Staubli VAL3: ToolItem.pjx

--- ToolItem.pjx ---
Parameters version=s7.2.1 stackSize=5000 millimeterUnit=true
Data file=toolItem.dtx
Type name=InstrItem path=Disk://kernel/template/InstrItem/InstrItem.pjx

--- ToolItem.dtx ---
public InstrItem iActionOFF[3]
  [0]
    string sType
    string sData
  [1]
    string sType
    string sData
  [2]
    string sType
    string sData
public InstrItem iActionON[3]
  [0]
    string sType
    string sData
  [1]
    string sType
    string sData
  [2]
    string sType
    string sData
public string name
public tool tcp = {fatherId=flange[0], ioLink=valve1}
